// TwinCAT 3 PLC project plc01
// ProgramVersion: 3.1.4026.24
// libraries:
//   Tc2_Standard, * (Beckhoff Automation GmbH)
//   Tc2_System, * (Beckhoff Automation GmbH)
//   Tc2_Utilities, * (Beckhoff Automation GmbH)
//   Tc3_Logging, * (www.peterzerlauth.com)
// project tree:
//   / FastTask.TcTTO, PlcTask.TcTTO
//   POUs/ FAST.TcPOU, FB_TestSlow.TcPOU, FB_TestFast.TcPOU, MAIN.TcPOU, POU.TcPOU (not stored)
// real-time tasks:
//   TASK SlowTask: cycle T#20ms, priority 20, ADS port 350
//   TASK FastTask: cycle T#1ms, priority 1, ADS port 351

CONFIGURATION plc01
    RESOURCE PLC ON TwinCAT3
        TASK FastTask(INTERVAL := T#1ms, PRIORITY := 1);
        TASK PlcTask(INTERVAL := T#20ms, PRIORITY := 20);
        PROGRAM FAST WITH FastTask : FAST;
        PROGRAM MAIN WITH PlcTask : MAIN;
    END_RESOURCE
END_CONFIGURATION

// ---- POUs/FAST.TcPOU
PROGRAM FAST
VAR
	fbTest:			FB_TestFast;
  	exception:			__SYSTEM.ExceptionCode;	
END_VAR

__TRY
	IF exception = __SYSTEM.ExceptionCode.RTSEXCPT_NOEXCEPTION THEN
		fbTest.P_Event.P_Logger:= MAIN.fbLogger;
	
	fbTest();
	
		
	END_IF


__CATCH(exception)


__ENDTRY

END_PROGRAM

// ---- POUs/FB_TestFast.TcPOU
FUNCTION_BLOCK FB_TestFast
VAR_INPUT
END_VAR
VAR_OUTPUT
END_VAR
VAR
	fbEvent: 			Tc3_Logging.FB_Event;
	bVerbose:			BOOL;
	bInfo:				BOOL;
	bWarning:			BOOL;
	bError:				BOOL;
	bCritical:			BOOL;

END_VAR

fbEvent();

// Demonstration of FB_Event usage with various log levels and argument types

IF bVerbose THEN
	fbEvent.P_Argument.M_AddINT(134052566194980000);
	fbEvent.P_Argument.M_AddSTRING('mm');
	fbEvent.M_Verbose('V message %s %s');
END_IF

IF bInfo THEN
	fbEvent.P_Argument.M_AddREAL(33.134581234, 3);
	fbEvent.P_Argument.M_AddSTRING('mm');
	fbEvent.M_Info('I message %s %s', 828536003);
END_IF

IF bWarning THEN
	fbEvent.M_Warning('W message', 475719253);
	fbEvent.M_Warning('W message', 475719253);
END_IF

IF bError THEN
	fbEvent.M_Error('E message', 475719235);
END_IF

IF bCritical THEN
	fbEvent.M_Critical('C message', 475719233);//475719234
	fbEvent.M_Critical('B message', 475719232); 
END_IF

PROPERTY PUBLIC P_Event : reference to FB_event
GET
P_Event ref= fbEvent;
END_GET
END_PROPERTY

END_FUNCTION_BLOCK

// ---- POUs/MAIN.TcPOU
PROGRAM MAIN
VAR
	fbLogger:			Tc3_Logging.FB_LoggerManager;
	fbHmiLogger:		Tc3_Logging.FB_HmiLogger;
	fbFileLogger:		Tc3_Logging.FB_FileLogger;
	fbTest:				FB_TestSlow;
  	exception:			__SYSTEM.ExceptionCode;	
	bReset: BOOL;
END_VAR

__TRY
	IF exception = __SYSTEM.ExceptionCode.RTSEXCPT_NOEXCEPTION THEN
		fbLogger.M_Add(fbHmiLogger);
		fbLogger.M_Add(fbFileLogger);
			
		fbHmiLogger();
		fbFileLogger.sPathName:= 'C:\temp\log.txt';
		fbFileLogger();

		
		
		IF bReset THEN
			fbTest.P_Event.M_Reset();
		END_IF
		
		fbTest.P_Event.P_Logger:= fbLogger;
		
		fbTest();	
		
// 		fbTest1000.P_Event.P_Logger:= fbLogger;
// 		fbTest1000();
		
	END_IF

__CATCH(exception)

__ENDTRY

END_PROGRAM

// ---- POUs/FB_TestSlow.TcPOU
FUNCTION_BLOCK FB_TestSlow
VAR_INPUT
END_VAR
VAR_OUTPUT
END_VAR
VAR
	fbEvent: 			Tc3_Logging.FB_Event;
	bVerbose:			BOOL;
	bInfo:				BOOL;
	bWarning:			BOOL;
	bError:				BOOL;
	bCritical:			BOOL;

END_VAR

fbEvent();

// Demonstration of FB_Event usage with various log levels and argument types

IF bVerbose THEN
	fbEvent.P_Argument.M_AddINT(134052566194980000);
	fbEvent.P_Argument.M_AddSTRING('mm');
	fbEvent.M_Verbose('V message %s %s');
END_IF

IF bInfo THEN
	fbEvent.P_Argument.M_AddREAL(33.0, 3);
	fbEvent.P_Argument.M_AddSTRING('mm');
	fbEvent.M_Info('I message %s %s', 828536003);
END_IF

IF bWarning THEN
	fbEvent.M_Warning('W message', 475719253);
	fbEvent.M_Warning('B message', 475719232);
	fbEvent.M_Warning('B messagex', 110769791);
	fbEvent.M_Warning('C messagex', 110769792);	
	fbEvent.M_Warning('X messagex', 110769813);	
END_IF


IF bError THEN
	fbEvent.M_Error('E message', 475719235);
END_IF

IF bCritical THEN
	fbEvent.M_Error('Input %s is simulated1', 361230260);
	fbEvent.M_Error('Input %s is simulated', 849363082);
	fbEvent.M_Error('Input %s is simulated2', 820656125);
	fbEvent.M_Error('Input %s is simulated2', 820656125);
END_IF

PROPERTY PUBLIC P_Event : reference to FB_event
GET
P_Event ref= fbEvent;
END_GET
END_PROPERTY

END_FUNCTION_BLOCK
